TYPE WMS_OPC_UA_DUT :
STRUCT
	Task_ID:  INT;
	Task_Metadata:  STRING[250];
	Task_Type:  Int;
	Source_Location:  DInt;
	Destination_Location:  DInt;
	Task_Data_Available:  Bool;
	SM_State:  UInt;
	Movement_Ready:  Bool;
	Movement_Request_Complete:  Bool;
	Movement_Request_Complete_Ack:  Bool;
	Shuttle_ID:  Int;
	Shuttle_Loaded:  Bool;
	Pallet_Type:  BYTE;
	Pallet_Alignment:  BYTE;
	SM_State_Maestro:  UInt;
	Pallet_Weight:  INT;
END_STRUCT
END_TYPE

(* stored: Version 1.1.0.1
   DUT WMS_OPC_UA_DUT: Id {8f9c193a-3459-4fcc-8c43-0ddf25e73618} *)
